{attribute addProperty BoxType "EL1512-0000-0016"}
{attribute addProperty Id "CNT_Inputs_ChannelAT %I*ARRAY[0..5] OF CNT_Inputs_Channel_445A37BE128160CNT_Outputs_ChannelAT %Q*ARRAY[0..3] OF CNT_Outputs_Channel_EEA87D4196120WcStateAT %I*WcState_98A4DF7520.250InfoDataAT %I*InfoData_BC63D37F80100"}
{attribute addProperty CRC "241302197"}
{attribute addProperty SizeInBites "306"}
{attribute addProperty SizeInBytes "38.25"}
TYPE EL1512_736E064C :
STRUCT
	{attribute addProperty Name "CNT_Inputs_Channel"}
	CNT_Inputs_Channel : ARRAY[0..5] OF CNT_Inputs_Channel_445A37BE;
	{attribute addProperty Name "CNT_Outputs_Channel"}
	CNT_Outputs_Channel : ARRAY[0..3] OF CNT_Outputs_Channel_EEA87D41;
	{attribute addProperty Name "WcState"}
	WcState : WcState_98A4DF75;
	{attribute addProperty Name "InfoData"}
	InfoData : InfoData_BC63D37F;
END_STRUCT
END_TYPE

(* stored: Version 1.2.0.0, ProductVersion 3.1.4024.9
   DUT EL1512_736E064C: Id {46af9615-a570-448b-96c7-7b4969e50521} *)
